// TIA Portal V20 export
// export: Created 2025-12-01T14:59:48.4511395Z, ExportSetting None, DisplayName Totally Integrated Automation Portal, DisplayVersion V20 Update 3, DisplayName TIA Portal Openness, DisplayVersion V20 Update 3, DisplayName TIA Portal Version Control Interface, DisplayVersion V20 Update 3, DisplayName STEP 7 Professional, DisplayVersion V20 Update 3, DisplayName STEP 7 Safety, DisplayVersion V20 Update 2, DisplayName WinCC Basic/Comfort/Advanced, DisplayVersion V20 Update 3, DisplayName WinCC Professional, DisplayVersion V20 Update 3, DisplayName WinCC Unified, DisplayVersion V20 Update 3
FUNCTION "FC400_Conector_TL_a_Mx" : Void   // FC400, LAD
{ S7_Optimized_Access := 'FALSE' }
AUTHOR : TLigero
NAME : 20130323
VERSION : 3.0
// stored: AutoNumber false, SetENOAutomatically false
   VAR_INPUT
      NumeroMesa_tracking : UInt;   // numero de mesa de la mesa de tracking
      PRV_AVTF : Bool;   // salida de la función de TL
      PRV_Descarga_Act : Bool;   // salida de la función TL
      NXT_PTF : Bool;   // Salida funcion tracking
      NXT_FTF : Bool;   // salida función tracking
   END_VAR
   VAR_OUTPUT
      PRV_CargaOK_Conector : Bool;   // marca que hay que llevar a la funcion de ligero
      PRV_Avance_Conector : Bool;   // marca que hay que llevar a la función de ligero
      NXT_AVTF_Conector : Bool;   // marca que hay que llevar a la función de tracking
   END_VAR
   VAR_IN_OUT
      NXT_DescargaAct_Conector : Bool;   // marca que hay que llevar a la función de tracking
   END_VAR
BEGIN

REGION Network 1: previo carga ok adaptacion a conectores
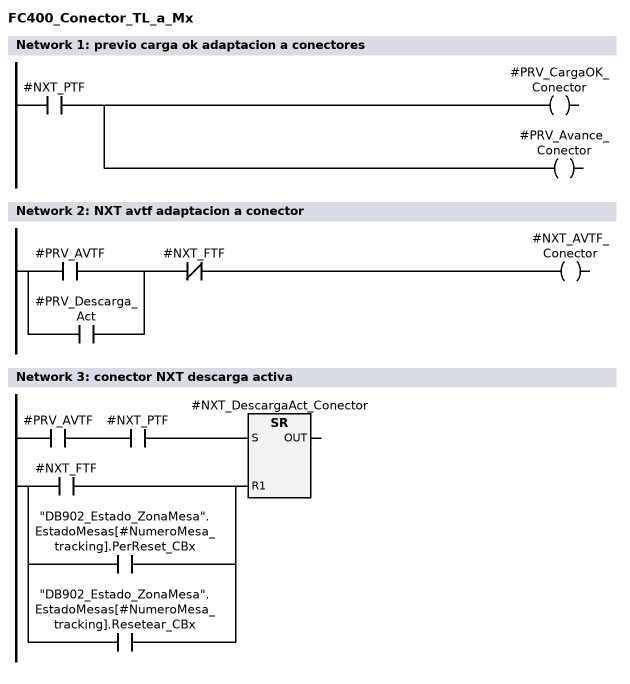
   RUNG wire#powerrail
      Contact( #NXT_PTF )
      wire#w1
      Coil( #PRV_CargaOK_Conector )
   END_RUNG
   RUNG wire#w1
      Coil( #PRV_Avance_Conector )
   END_RUNG
   // the same network as SCL:
   #PRV_CargaOK_Conector := #NXT_PTF;
   #PRV_Avance_Conector := #NXT_PTF;
END_REGION

REGION Network 2: NXT avtf adaptacion a conector
   RUNG wire#powerrail
      Contact( #PRV_AVTF )
      wire#w1
      I_Contact( #NXT_FTF )
      Coil( #NXT_AVTF_Conector )
   END_RUNG
   RUNG wire#powerrail
      Contact( #PRV_Descarga_Act )
   END_RUNG wire#w1
   // the same network as SCL:
   #NXT_AVTF_Conector := (#PRV_AVTF OR #PRV_Descarga_Act) AND NOT #NXT_FTF;
END_REGION

REGION Network 3: conector NXT descarga activa
   RUNG wire#powerrail
      Contact( #PRV_AVTF )
      Contact( #NXT_PTF )
      S_SR(operand := #NXT_DescargaAct_Conector, r1 := wire#w1)
   END_RUNG
   RUNG wire#powerrail
      Contact( #NXT_FTF )
   END_RUNG wire#w1
   RUNG wire#powerrail
      Contact( "DB902_Estado_ZonaMesa".EstadoMesas[#NumeroMesa_tracking].PerReset_CBx )
   END_RUNG wire#w1
   RUNG wire#powerrail
      Contact( "DB902_Estado_ZonaMesa".EstadoMesas[#NumeroMesa_tracking].Resetear_CBx )
   END_RUNG wire#w1
   // the same network as SCL:
   IF #PRV_AVTF AND #NXT_PTF THEN
       #NXT_DescargaAct_Conector := TRUE;   // SR flip-flop
   END_IF;
   IF #NXT_FTF OR "DB902_Estado_ZonaMesa".EstadoMesas[#NumeroMesa_tracking].PerReset_CBx OR "DB902_Estado_ZonaMesa".EstadoMesas[#NumeroMesa_tracking].Resetear_CBx THEN
       #NXT_DescargaAct_Conector := FALSE;
   END_IF;
END_REGION
END_FUNCTION
